VAR_GLOBAL
	bLimitForward AT %Q* : BOOL := TRUE;
	bLimitBackward AT %Q* : BOOL := TRUE;

	eStageEnableMode : ENUM_StageEnableMode := ENUM_StageEnableMode.ALWAYS;
    {attribute 'TcLinkTo' := '.bLimitForwardEnable  := TIPC^test_cablelength^test_cablelength Instance^PlcTask Outputs^GVL_Devices.bLimitForward;
                              .bLimitBackwardEnable := TIPC^test_cablelength^test_cablelength Instance^PlcTask Outputs^GVL_Devices.bLimitBackward;
							  .nRawEncoderULINT     := TIIB[Term 3 (EL5042)]^FB Inputs Channel 2^Position'}
    {attribute 'pytmc' := '
        pv: TST:LAB:MMS:01
    '}
    M1: ST_MotionStage := (
        bHardwareEnable := TRUE,
        bPowerSelf := TRUE,	
        nEnableMode := eStageEnableMode,
        nHomingMode := ENUM_EpicsHomeCmd.NONE,
        sName := 'TST:LAB:MMS:01');
	(*.bLimitForwardEnable  := TIIB[Term 2 (EL7047)]^STM Status^Status^Digital input 1;
                              .bLimitBackwardEnable := TIIB[Term 2 (EL7047)]^STM Status^Status^Digital input 2;*)
							  
END_VAR

(* stored: Version 1.1.0.1, ProductVersion 3.1.4022.18
   GVL GVL_Devices: Id {e3833f14-22ee-49ed-9099-87e4ce64c3f5} *)
